{attribute 'qualified_only'}
TYPE E_LockCtrl :
(
	Unlock,
	Lock
)USINT;
END_TYPE

(* stored: Version 1.1.0.1, ProductVersion 3.1.4024.11
   DUT E_LockCtrl: Id {220e2e51-4335-47c0-874b-f128028fdbc2} *)
